% RSLogix 500 project DIGITAL_CONTROL_LOGIC.RSS, saved by version 8.30.00.16 %
PROJECT "PROC1"    % processor: Bul.1763 MicroLogix 1100 Series B %

PROGRAM FILES
  LAD 2 "MAIN"  3 rungs
  LAD 3 "IO"  5 rungs
  LAD 4 "CONTROLS"  11 rungs

DATA FILES
  O0 OUTPUT  4 elements
  I1 INPUT  6 elements
  S2 STATUS  66 elements
  B3 BINARY  1 elements
  T4 TIMER  4 elements
  C5 COUNTER  1 elements
  R6 CONTROL  1 elements
  N7 INTEGER  1 elements
  F8 FLOAT  1 elements

LADDER 2 "MAIN"
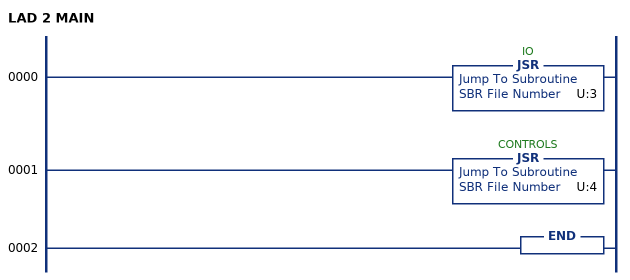
% Rung: 0 %
SOR JSR U:3 EOR
%   U:3  "IO" %
% Rung: 1 %
SOR JSR U:4 EOR
%   U:4  "CONTROLS" %
% Rung: 2 %
SOR END EOR

LADDER 3 "IO"
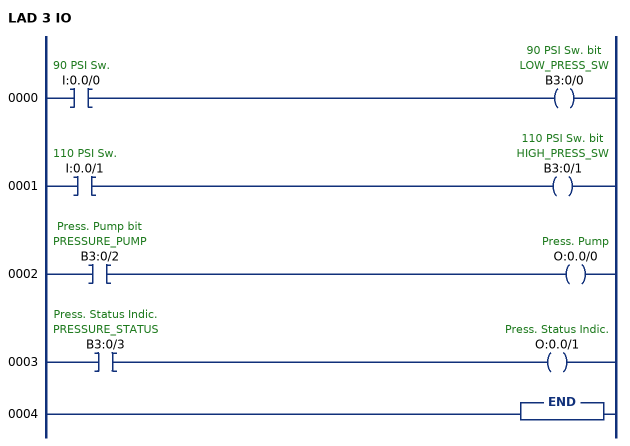
% Rung: 0 %
SOR XIC I:0.0/0 OTE B3:0/0 EOR
%   I:0.0/0  "90 PSI Sw." %
%   B3:0/0  LOW_PRESS_SW  "90 PSI Sw. bit" %
% Rung: 1 %
SOR XIC I:0.0/1 OTE B3:0/1 EOR
%   I:0.0/1  "110 PSI Sw." %
%   B3:0/1  HIGH_PRESS_SW  "110 PSI Sw. bit" %
% Rung: 2 %
SOR XIC B3:0/2 OTE O:0.0/0 EOR
%   B3:0/2  PRESSURE_PUMP  "Press. Pump bit" %
%   O:0.0/0  "Press. Pump" %
% Rung: 3 %
SOR XIC B3:0/3 OTE O:0.0/1 EOR
%   B3:0/3  PRESSURE_STATUS  "Press. Status Indic." %
%   O:0.0/1  "Press. Status Indic." %
% Rung: 4 %
SOR END EOR

LADDER 4 "CONTROLS"
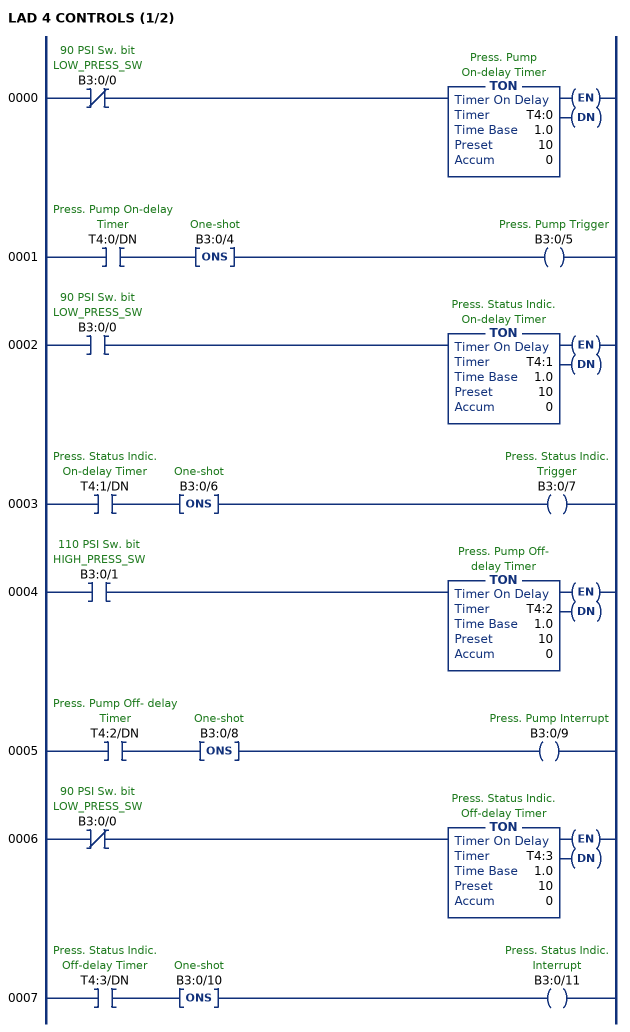
% Rung: 0 %
SOR XIO B3:0/0 TON T4:0 1.0 10 0 EOR
%   B3:0/0  LOW_PRESS_SW  "90 PSI Sw. bit" %
%   T4:0  "Press. Pump On-delay Timer" %
% Rung: 1 %
SOR XIC T4:0/DN ONS B3:0/4 OTE B3:0/5 EOR
%   T4:0  "Press. Pump On-delay Timer" %
%   B3:0/4  "One-shot" %
%   B3:0/5  "Press. Pump Trigger" %
% Rung: 2 %
SOR XIC B3:0/0 TON T4:1 1.0 10 0 EOR
%   B3:0/0  LOW_PRESS_SW  "90 PSI Sw. bit" %
%   T4:1  "Press. Status Indic. On-delay Timer" %
% Rung: 3 %
SOR XIC T4:1/DN ONS B3:0/6 OTE B3:0/7 EOR
%   T4:1  "Press. Status Indic. On-delay Timer" %
%   B3:0/6  "One-shot" %
%   B3:0/7  "Press. Status Indic. Trigger" %
% Rung: 4 %
SOR XIC B3:0/1 TON T4:2 1.0 10 0 EOR
%   B3:0/1  HIGH_PRESS_SW  "110 PSI Sw. bit" %
%   T4:2  "Press. Pump Off- delay Timer" %
% Rung: 5 %
SOR XIC T4:2/DN ONS B3:0/8 OTE B3:0/9 EOR
%   T4:2  "Press. Pump Off- delay Timer" %
%   B3:0/8  "One-shot" %
%   B3:0/9  "Press. Pump Interrupt" %
% Rung: 6 %
SOR XIO B3:0/0 TON T4:3 1.0 10 0 EOR
%   B3:0/0  LOW_PRESS_SW  "90 PSI Sw. bit" %
%   T4:3  "Press. Status Indic. Off-delay Timer" %
% Rung: 7 %
SOR XIC T4:3/DN ONS B3:0/10 OTE B3:0/11 EOR
%   T4:3  "Press. Status Indic. Off-delay Timer" %
%   B3:0/10  "One-shot" %
%   B3:0/11  "Press. Status Indic. Interrupt" %

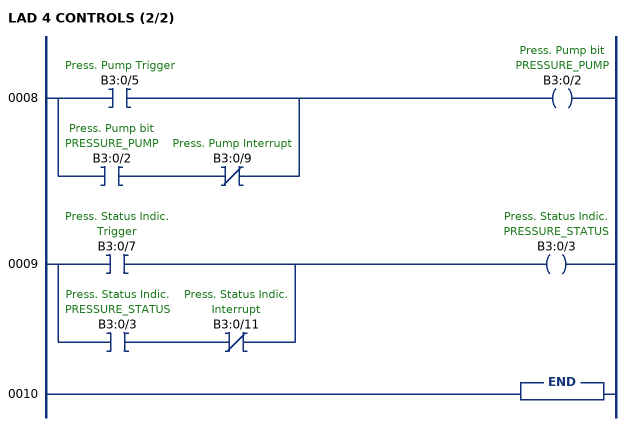
% Rung: 8 %
SOR BST XIC B3:0/5 NXB XIC B3:0/2 XIO B3:0/9 BND OTE B3:0/2 EOR
%   B3:0/5  "Press. Pump Trigger" %
%   B3:0/2  PRESSURE_PUMP  "Press. Pump bit" %
%   B3:0/9  "Press. Pump Interrupt" %
% Rung: 9 %
SOR BST XIC B3:0/7 NXB XIC B3:0/3 XIO B3:0/11 BND OTE B3:0/3 EOR
%   B3:0/7  "Press. Status Indic. Trigger" %
%   B3:0/3  PRESSURE_STATUS  "Press. Status Indic." %
%   B3:0/11  "Press. Status Indic. Interrupt" %
% Rung: 10 %
SOR END EOR

DATA TABLE (non-zero values as saved)
DATA T4
% .PRE .ACC %
% T4:0 % 10 0
% T4:1 % 10 0
% T4:2 % 10 0
% T4:3 % 10 0
